FUNCTION_BLOCK EffluentSensors (* CAT Function Block Type *)
  (* Standard: 61499-2 *)
  (* Version 0.0, 6/13/2026, Schneider Electric, template *)
  PACKAGE SE.Nereda;
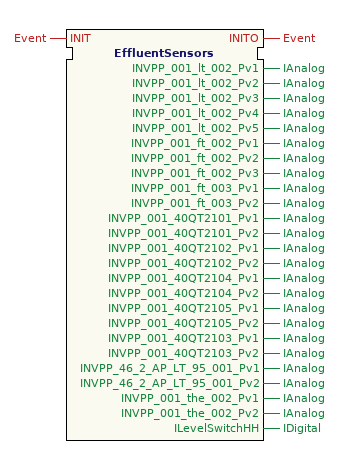
  EVENT_INPUT
    INIT; (* Initializes the symbolic link data destination FB with N (1 <= N <= 16) variables *)
  END_EVENT
  EVENT_OUTPUT
    INITO; (* Initialization Confirm *)
  END_EVENT
  PLUGS
    INVPP_001_lt_002_Pv1 : IAnalog; (* Process value and status interface adapter *)
    INVPP_001_lt_002_Pv2 : IAnalog; (* Process value and status interface adapter *)
    INVPP_001_lt_002_Pv3 : IAnalog; (* Process value and status interface adapter *)
    INVPP_001_lt_002_Pv4 : IAnalog; (* Process value and status interface adapter *)
    INVPP_001_lt_002_Pv5 : IAnalog; (* Process value and status interface adapter *)
    INVPP_001_ft_002_Pv1 : IAnalog; (* Process value and status interface adapter *)
    INVPP_001_ft_002_Pv2 : IAnalog; (* Process value and status interface adapter *)
    INVPP_001_ft_002_Pv3 : IAnalog; (* Process value and status interface adapter *)
    INVPP_001_ft_003_Pv1 : IAnalog; (* Process value and status interface adapter *)
    INVPP_001_ft_003_Pv2 : IAnalog; (* Process value and status interface adapter *)
    INVPP_001_40QT2101_Pv1 : IAnalog; (* Process value and status interface adapter *)
    INVPP_001_40QT2101_Pv2 : IAnalog; (* Process value and status interface adapter *)
    INVPP_001_40QT2102_Pv1 : IAnalog; (* Process value and status interface adapter *)
    INVPP_001_40QT2102_Pv2 : IAnalog; (* Process value and status interface adapter *)
    INVPP_001_40QT2104_Pv1 : IAnalog; (* Process value and status interface adapter *)
    INVPP_001_40QT2104_Pv2 : IAnalog; (* Process value and status interface adapter *)
    INVPP_001_40QT2105_Pv1 : IAnalog; (* Process value and status interface adapter *)
    INVPP_001_40QT2105_Pv2 : IAnalog; (* Process value and status interface adapter *)
    INVPP_001_40QT2103_Pv1 : IAnalog; (* Process value and status interface adapter *)
    INVPP_001_40QT2103_Pv2 : IAnalog; (* Process value and status interface adapter *)
    INVPP_46_2_AP_LT_95_001_Pv1 : IAnalog; (* Process value and status interface adapter *)
    INVPP_46_2_AP_LT_95_001_Pv2 : IAnalog; (* Process value and status interface adapter *)
    INVPP_001_the_002_Pv1 : IAnalog; (* Process value and status interface adapter *)
    INVPP_001_the_002_Pv2 : IAnalog; (* Process value and status interface adapter *)
    ILevelSwitchHH : IDigital; (* Process value interface adapter *)
  END_PLUGS
  (* 01 - FUNCTIONNAL INPUT INTERFACE *)
  (* 00 - INITIALIZATION *)
  (* 05 - LOGIC *)
  (* 06 - HMI INTERFACE *)
  (* 02 - FUNCTIONNAL OUTPUT INTERFACE *)
  (* Sensors Status *)
  (* 03 - FIELD INTERFACE *)
  (* Turbidity/dry solids measurement effluent *)
  (* Phosphate PO4 measurement effluent *)
  (* Ammonium NH4 measurement *)
  (* Nitrate NO3 measurement *)
  (* Auto sampler *)
  (* Flow measurement effluent *)
  (* Tertiary filter flow *)
  (* Level Sensor Effluent *)
  (* Level Sensor Calamity *)
  (* Ambient temperature *)
  FBS
    TurbidityMeasurementEffluent_Status : AnalogInput_Status;
    NVPP_001_40QT2102_Status : AnalogInput_Status;
    NVPP_001_40QT2104_Status : AnalogInput_Status;
    TurbidityMeasurementEffluent : AnalogInput;
    NVPP_001_40QT2102 : AnalogInput;
    NVPP_001_40QT2104 : AnalogInput;
    HiLevelSwitch_Calamity : DigitalInput;
    NVPP_001_40QT2105 : AnalogInput;
    NVPP_001_40QT2103 : AnalogInput;
    NVPP_001_ft_002 : AnalogInput;
    NVPP_001_ft_003 : AnalogInput;
    NVPP_001_lt_002 : AnalogInput;
    NVPP_46_2_AP_LT_95_001 : AnalogInput;
    NVPP_001_the_002 : AnalogInput;
    NVPP_001_40QT2105_Status : AnalogInput_Status;
    NVPP_001_40QT2103_Status : AnalogInput_Status;
    NVPP_001_ft_002_Status : AnalogInput_Status;
    NVPP_001_ft_003_Status : AnalogInput_Status;
    NVPP_001_lt_002_Status : AnalogInput_Status;
    NVPP_46_2_AP_LT_95_001_Status : AnalogInput_Status;
    NVPP_001_the_002_Status : AnalogInput_Status;
  END_FBS
  EVENT_CONNECTIONS
    INIT TO TurbidityMeasurementEffluent_Status.INIT;
    TurbidityMeasurementEffluent_Status.INITO TO NVPP_001_40QT2102_Status.INIT;
    NVPP_001_40QT2102_Status.INITO TO NVPP_001_40QT2104_Status.INIT;
    NVPP_001_40QT2104_Status.INITO TO NVPP_001_40QT2105_Status.INIT;
    NVPP_001_40QT2105_Status.INITO TO NVPP_001_40QT2103_Status.INIT;
    NVPP_001_40QT2103_Status.INITO TO NVPP_001_ft_002_Status.INIT;
    NVPP_001_ft_002_Status.INITO TO NVPP_001_ft_003_Status.INIT;
    NVPP_001_ft_003_Status.INITO TO NVPP_001_lt_002_Status.INIT;
    NVPP_001_lt_002_Status.INITO TO NVPP_46_2_AP_LT_95_001_Status.INIT;
    NVPP_46_2_AP_LT_95_001_Status.INITO TO NVPP_001_the_002_Status.INIT;
    NVPP_001_the_002_Status.INITO TO INITO;
  END_CONNECTIONS
  ADAPTER_CONNECTIONS
    TurbidityMeasurementEffluent.73A667132981F8F7 TO TurbidityMeasurementEffluent_Status.404867D502801067;
    TurbidityMeasurementEffluent.5EC3A1C2B6EC87E8 TO INVPP_001_40QT2101_Pv1;
    TurbidityMeasurementEffluent.95FA69AE12D9BDE1 TO INVPP_001_40QT2101_Pv2;
    NVPP_001_40QT2102.73A667132981F8F7 TO NVPP_001_40QT2102_Status.404867D502801067;
    NVPP_001_40QT2102.5EC3A1C2B6EC87E8 TO INVPP_001_40QT2102_Pv1;
    NVPP_001_40QT2102.95FA69AE12D9BDE1 TO INVPP_001_40QT2102_Pv2;
    NVPP_001_40QT2104.73A667132981F8F7 TO NVPP_001_40QT2104_Status.404867D502801067;
    NVPP_001_40QT2104.5EC3A1C2B6EC87E8 TO INVPP_001_40QT2104_Pv1;
    NVPP_001_40QT2104.95FA69AE12D9BDE1 TO INVPP_001_40QT2104_Pv2;
    HiLevelSwitch_Calamity.252883A7B7227472 TO ILevelSwitchHH;
    NVPP_001_40QT2105.5EC3A1C2B6EC87E8 TO INVPP_001_40QT2105_Pv1;
    NVPP_001_40QT2105.95FA69AE12D9BDE1 TO INVPP_001_40QT2105_Pv2;
    NVPP_001_40QT2103.5EC3A1C2B6EC87E8 TO INVPP_001_40QT2103_Pv1;
    NVPP_001_40QT2103.95FA69AE12D9BDE1 TO INVPP_001_40QT2103_Pv2;
    NVPP_001_ft_002.5EC3A1C2B6EC87E8 TO INVPP_001_ft_002_Pv1;
    NVPP_001_ft_002.95FA69AE12D9BDE1 TO INVPP_001_ft_002_Pv2;
    NVPP_001_ft_002.84357DECBC9FC157 TO INVPP_001_ft_002_Pv3;
    NVPP_001_ft_003.5EC3A1C2B6EC87E8 TO INVPP_001_ft_003_Pv1;
    NVPP_001_ft_003.95FA69AE12D9BDE1 TO INVPP_001_ft_003_Pv2;
    NVPP_001_lt_002.5EC3A1C2B6EC87E8 TO INVPP_001_lt_002_Pv1;
    NVPP_001_lt_002.95FA69AE12D9BDE1 TO INVPP_001_lt_002_Pv2;
    NVPP_001_lt_002.84357DECBC9FC157 TO INVPP_001_lt_002_Pv3;
    NVPP_001_lt_002.0D7BD97A245CBD60 TO INVPP_001_lt_002_Pv4;
    NVPP_001_lt_002.6EF0614AFA3F1863 TO INVPP_001_lt_002_Pv5;
    NVPP_46_2_AP_LT_95_001.5EC3A1C2B6EC87E8 TO INVPP_46_2_AP_LT_95_001_Pv1;
    NVPP_46_2_AP_LT_95_001.95FA69AE12D9BDE1 TO INVPP_46_2_AP_LT_95_001_Pv2;
    NVPP_001_the_002.5EC3A1C2B6EC87E8 TO INVPP_001_the_002_Pv1;
    NVPP_001_the_002.95FA69AE12D9BDE1 TO INVPP_001_the_002_Pv2;
    NVPP_001_40QT2105.73A667132981F8F7 TO NVPP_001_40QT2105_Status.404867D502801067;
    NVPP_001_40QT2103.73A667132981F8F7 TO NVPP_001_40QT2103_Status.404867D502801067;
    NVPP_001_ft_002.73A667132981F8F7 TO NVPP_001_ft_002_Status.404867D502801067;
    NVPP_001_ft_003.73A667132981F8F7 TO NVPP_001_ft_003_Status.404867D502801067;
    NVPP_001_lt_002.73A667132981F8F7 TO NVPP_001_lt_002_Status.404867D502801067;
    NVPP_46_2_AP_LT_95_001.73A667132981F8F7 TO NVPP_46_2_AP_LT_95_001_Status.404867D502801067;
    NVPP_001_the_002.73A667132981F8F7 TO NVPP_001_the_002_Status.404867D502801067;
  END_CONNECTIONS
END_FUNCTION_BLOCK
